FUNCTION F_GetPumpPath : E_PumpPath
VAR_INPUT
	iValvePosition	: SINT;
	ePumpDirection	: E_PumpDirection;
END_VAR
VAR
END_VAR

CASE iValvePosition OF
	
	1:
		F_GetPumpPath := E_PumpPath.FillJars;
		RETURN;
	
	2:
		F_GetPumpPath := E_PumpPath.FillJars;
		RETURN;
	
	3:
		F_GetPumpPath := E_PumpPath.FillJars;
		RETURN;
		
	4:
		F_GetPumpPath := E_PumpPath.FillJars;
		RETURN;
		
	5:
		F_GetPumpPath := E_PumpPath.FillCalBox;
		RETURN;
	6:
		IF ePumpDirection = E_PumpDirection.Forward THEN
			F_GetPumpPath := E_PumpPath.FromCalBox;
			RETURN;
			ELSIF ePumpDirection = E_PumpDirection.Backward THEN
				F_GetPumpPath := E_PumpPath.FillCalBox;
				RETURN;
		ELSE
			F_GetPumpPath := E_PumpPath.FromCalBox;
			RETURN;
		END_IF

END_CASE

END_FUNCTION

(* stored: Version 1.1.0.1, ProductVersion 3.1.4024.12
   POU F_GetPumpPath: Id {da8f6142-46aa-4ab1-9d35-c600d380a07e}, SpecialFunc None *)
